// TIA Portal V17 export
// export: Created 2026-05-13T16:54:41.5834471Z, ExportSetting WithDefaults, DisplayName Totally Integrated Automation Portal, DisplayVersion V17 Update 4, DisplayName TIA Portal Openness, DisplayVersion V17 Update 4, DisplayName TIA Portal Version Control Interface, DisplayVersion V17, DisplayName SINAMICS Startdrive Advanced, DisplayVersion V17, DisplayName SINAMICS Startdrive G130, G150, S120, S150, SINAMICS MV, S210, DisplayVersion V17, DisplayName SINAMICS Startdrive G110M, G120, G120C, G120D, G120P, G115D, DisplayVersion V17, DisplayName STEP 7 Professional, DisplayVersion V17 Update 4, DisplayName STEP 7 Safety, DisplayVersion V17, DisplayName WinCC Professional, DisplayVersion V17 Update 4
TagTable "M"
  MZT主塔气扫 : Bool  (PLC tag MZT主塔气扫, HMI_连接_1, 1 s)
  MBD布袋反吹 : Bool  (PLC tag MBD布袋反吹, HMI_连接_1, 1 s)
  MZT主塔振打 : Bool  (PLC tag MZT主塔振打, HMI_连接_1, 1 s)
  MJL进料泵 : Bool  (PLC tag MJL进料泵, HMI_连接_1, 1 s)
  MJL进料泵正反转 : Bool  (PLC tag MJL进料泵正反转, HMI_连接_1, 1 s)
  MDJ电加热 : Bool  (PLC tag MDJ电加热, HMI_连接_1, 1 s)
  MZM照明灯 : Bool  (PLC tag MZM照明灯, HMI_连接_1, 1 s)
  MAQ安全停机 : Bool  (PLC tag MAQ安全停机, HMI_连接_1, 1 s)
  MJF进温自整定 : Bool  (PLC tag MJF进温自整定, HMI_连接_1, 1 s)
  MYF引风机 : Bool  (PLC tag MYF引风机, HMI_连接_1, 1 s)
  MLX离心雾化 : Bool  (PLC tag MLX离心雾化, HMI_连接_1, 1 s)
  MBD布袋振打 : Bool  (PLC tag MBD布袋振打, HMI_连接_1, 1 s)
  MZM照明 : Bool  (PLC tag MZM照明, HMI_连接_1, 1 s)
  MHW恒温系统 : Bool  (PLC tag MHW恒温系统, HMI_连接_1, 1 s)
  MRS热水炉 : Bool  (PLC tag MRS热水炉, HMI_连接_1, 1 s)
  MRS热水炉自整定 : Bool  (PLC tag MRS热水炉自整定, HMI_连接_1, 1 s)
  MQL气离切换 : Bool  (PLC tag MQL气离切换, HMI_连接_1, 1 s)
